(* PLC project Generated.project, CODESYS CODESYS V3.5 SP19 Patch 1 *)
(* stored: creationDateTime 2026-08-19T02:05:17.219400, modificationDateTime 2026-08-19T02:05:17.219400 *)

(* ═══════════════════════════════════════════════════════════════ 🌐 ST_BypassNetwork — Bypass général du diagnostic réseau ─────────────────────────────────────────────────────────────── 🔒 Permet de forcer les esclaves réseau (CAN, EtherCAT) à "online" pour le diagnostic, sans devoir toucher à chaque bit individuel. Jamais actif en production. ═══════════════════════════════════════════════════════════════ *)
TYPE ST_BypassNetwork : STRUCT
  Joystick : BOOL;  (* 📡 1. Communication & Systèmes esclaves 🕹️ Bypass diagnostic esclave CANopen Joystick *)
  EncoderM1 : BOOL;  (* 🧲 Bypass diagnostic esclave EtherCAT COD1 (M1 codeur) *)
  EncoderM2 : BOOL;  (* 🧲 Bypass diagnostic esclave EtherCAT COD2 (M2 codeur) *)
  VariateurM3 : BOOL;  (* ↔️ Bypass diagnostic esclave EtherCAT AC600 (M3 drive) *)
  IhmHeartbeat : BOOL := TRUE;  (* 💓 Bypass du bit de vie IHM (défaut TRUE = sécurisé si pas d'IHM) *)
  Global : BOOL;  (* 🛡️ 2. Hiérarchie & Restauration 🌐 Bypass Global : tous les esclaves réseau à la fois *)
  Initialized : BOOL := FALSE;  (* Flag restauration boot dédié (défaut FALSE non ambigu, contrairement à une valeur métier) 🚦 TRUE = bypass restauré depuis GVL_BypassRetain ce boot *)
END_STRUCT;
END_TYPE
